# EPICS autosave request: ADApp/Db/pilatus_settings.req
$(P)$(R)DelayTime
$(P)$(R)ThresholdEnergy
$(P)$(R)GainMenu
$(P)$(R)ReadTiffTimeout
$(P)$(R)BadPixelFile
$(P)$(R)FlatFieldFile
$(P)$(R)MinFlatField
